// TIA Portal V16 export
// export: Created 2023-10-30T22:43:55.8879423Z, ExportSetting WithDefaults, DisplayName Totally Integrated Automation Portal, DisplayVersion V16, DisplayName TIA Portal Version Control Interface, DisplayVersion V16, DisplayName TIA Portal Openness, DisplayVersion V16, DisplayName SINAMICS Startdrive Advanced, DisplayVersion V16, DisplayName SINAMICS Startdrive G130, G150, S120, S150, SINAMICS MV, S210, DisplayVersion V16, DisplayName SINAMICS Startdrive G110M, G120, G120C, G120D, G120P, DisplayVersion V16, DisplayName STEP 7 Professional, DisplayVersion V16, DisplayName STEP 7 Safety, DisplayVersion V16, DisplayName WinCC Professional, DisplayVersion V16
DATA_BLOCK "Simulacion_HR_DB"   // DB23
VERSION : 0.1
// stored: AutoNumber true, DBAccessibleFromOPCUA true, InstanceOfName Simulacion_HR, InstanceOfType FB
"Simulacion_HR"
   // VAR_OUTPUT
   //    y3 : Int;
   // END_VAR
   // VAR
   //    Timer_SimHR : Struct
   //       IN : Bool;
   //       PT : Time;
   //       Q : Bool;
   //       ET : Time;
   //    END_STRUCT;
   //    t : Int;
   //    t2 : Real;
   //    y3_Aux : Int;
   // END_VAR
BEGIN
END_DATA_BLOCK
